(*
SPDX-FileCopyrightText: © 2026 Oleksandr Tiutyk <trofimich@gmail.com>
SPDX-License-Identifier: MIT
License: https://opensource.org/license/mit
*)

(*!
<summary>Reports an unassigned required reference.</summary>
<description>
The caller detects the missing reference before dereferencing it. This exception records its name; it does not
inspect memory or test object lifetime. Uses the GeneralException task-local cycle lifetime and throw rules.
Dynamic copies are explicitly registered by Clone after construction; plain __NEW does not transfer ownership
to the task manager.
</description>
*)

{attribute 'enable_dynamic_creation'}
{attribute 'no_explicit_call' := 'do not call this function block directly'}
FUNCTION_BLOCK NullReferenceException EXTENDS GeneralException IMPLEMENTS INullReferenceException
VAR_STAT
	//! <summary>Class name shared by all instances of this function block.</summary>
	{attribute 'hide'} 
	_ClassName : STRING := __POUNAME();
END_VAR

{attribute 'monitoring' := 'call'}
PROPERTY ClassName : REFERENCE TO STRING
GET
ClassName REF= _ClassName;
END_GET
END_PROPERTY

(*!
<summary>Creates a clone of this concrete exception type.</summary>
<description>
Copies GeneralException fields and timestamps. DynamicMemoryManager owns the clone until cleanup of the
creating task; callers must not delete it. Allocation failure is terminal. Registers the newly constructed
instance before copying payload, outside FB_init. Registration failure releases the unregistered instance and
raises a terminal error; copy failure leaves the registered instance owned by the task manager for cleanup.
Custom overrides must follow the same ownership sequence.
</description>
*)
METHOD Clone : IObject
VAR
	exceptionClone : POINTER TO NullReferenceException;
END_VAR
exceptionClone := __NEW(NullReferenceException);

IF exceptionClone = 0 THEN
	DynamicMemoryManager.RaiseAllocationFailure();
END_IF

DynamicMemoryManager.RegisterAutoDisposedObject(autoDisposedObject := exceptionClone^);

exceptionClone^.CopyGeneralFields(sourceException := THIS^);

Clone := exceptionClone^;
END_METHOD

(*!
<summary>Provides the library namespace used in diagnostics.</summary>
<description>
Borrowed read-only reference to the compiler-initialized library namespace; no ownership transfer.
</description>
*)
{attribute 'monitoring' := 'call'}
PROPERTY NamespaceName : REFERENCE TO STRING
GET
NamespaceName REF= CurrentNamespace.Name;
END_GET
END_PROPERTY

(*!
<summary>Reports the byte size of this concrete instance.</summary>
<description>
Uses XSIZEOF on the instance. Does not include separately allocated payloads or prove that an arbitrary
address is valid.
</description>
*)
{attribute 'monitoring' := 'call'}
PROPERTY SelfSize : ULINT
GET
SelfSize := XSIZEOF(THIS^);
END_GET
END_PROPERTY

(*!
<summary>Reports the missing reference and raises this exception.</summary>
<description>
Sets error code to zero and supplies no inner exception. Call only in cyclic task context, not during FB_init.
</description>
<param name="variableOrPropertyName">Name of the required variable or property that is not assigned.</param>
*)
METHOD Throw
VAR_INPUT
	sourceNamespaceName : STRING;
	sourceClassName : STRING;
	sourcePOUName : STRING;
	sourcePosition : STRING;
	variableOrPropertyName : STRING;
END_VAR
VAR
	message : ERROR_MESSAGE;
END_VAR
message := WideStrings.Concat255("Required reference '", TO_WSTRING(variableOrPropertyName), "' is not assigned");

InternalThrow(
	sourceNamespaceName := sourceNamespaceName,
	sourceClassName := sourceClassName,
	sourcePOUName := sourcePOUName,
	sourcePosition := sourcePosition,
	message := message,
	errorCode := 0,
	innerException := 0
);
END_METHOD

END_FUNCTION_BLOCK

(* stored: Version 1.1.0.1
   POU NullReferenceException: Id {652b5f52-6cdf-48c1-95a9-e9e566565f3b}, SpecialFunc None
   Property ClassName: Id {c372a7a1-140f-4ef6-9336-183c32e58e3d}
   Get Get: Id {9a9e6dda-c880-4ae7-a7ec-959ab6c26e77}
   Method Clone: Id {3a60293e-78ab-4fed-ba6d-7b196c7a0582}
   Property NamespaceName: Id {040c85e8-ee23-44b3-82cf-533c9538a2bf}
   Get Get: Id {43b74174-18e2-49f5-a856-c7db31f5844a}
   Property SelfSize: Id {7bf52448-f186-4337-9db3-2658a576f1d6}
   Get Get: Id {b52f1297-ecf9-4f60-be3a-53f670420c23}
   Method Throw: Id {b678bf91-26d4-49b0-bddd-ab608bfbc708} *)
